Fanuc KAREL source: kt00589.KL

-- PROVISIONAL review KL for V770-1; original PC SHA256 fbad1f32fce0e547f34de8c0e5e6b4474cf06e45546321c92ae789e7d18d4a50
-- Incomplete behavior may be omitted. Consult companion uncertainty JSON. Do not deploy.
PROGRAM KT00589
%NOLOCKGROUP
VAR
  S1 : STRING[80]
  S2 : STRING[80]
  OUT : STRING[80]
BEGIN
  -- UNRESOLVED_PC offsets 5-14; opcodes 3F,75
  -- UNRESOLVED_PC offsets 19-28; opcodes 3F,75
  -- UNRESOLVED_PC offsets 33-42; opcodes 3F,75
  -- UNRESOLVED_PC offsets 47-56; opcodes 3F,75
  -- UNRESOLVED_PC offsets 61-80; opcodes 73,73,7D,75
  -- UNRESOLVED_PC offsets 85-89; opcodes 7F
END KT00589
